KUKA KRL program: WL_TASMOCIAG_TIMER.src

&ACCESS RVO1
&COMMENT
DEF WL_TASMOCIAG_TIMER (CZY_WLACZYC :IN)

BOOL CZY_WLACZYC

WL_TIMER(CZY_WLACZYC)
WL_TASMOCIAG(CZY_WLACZYC)

END
